// TIA Portal V18 export
DATA_BLOCK "HMI"   // DB1
{ S7_Optimized_Access := 'TRUE' }
VERSION : 0.1
// stored: AutoNumber true, DBAccessibleFromOPCUA true, IsOnlyStoredInLoadMemory false, IsRetainMemResEnabled false, IsWriteProtectedInAS false, MemoryReserve 100
   VAR
      "screen no to change" : Int;
      unit : Struct
         cm3 : Int;
         cm3_min : Int;
         ml : Int;
         ml_min : Int;
         "degree celsius" : Int;
         precentage : Int;
         seonds : Int;
         minutes : Int;
         hours : Int;
         bar : Int;
         mbar : Int;
         milliseconds : Int;
         RPM : Int;
         imp : Int;
         "cm3/r" : Int;
         set : Int;
         "real" : Int;
         "type" : Int;
         day : Int;
         "cm3/imp" : Int;
         "imp/rev" : Int;
         "m" : Int;
      END_STRUCT;
      "A" : Int;
      "B" : Int;
      "Screen no by function" : Int;
      "Current screen No" : Int;
      "Function ONS" : Struct
         "Dearing A" : Bool;
         "function deselected" : Bool;
         "Dearing B" : Bool;
         "Dearing A coil" : Bool;
         "dearing B Coil" : Bool;
         Flush : Bool;
         "pre run" : Bool;
         "Ratio Check" : Bool;
         "Shot metering Program" : Bool;
         "Continous metering prgram" : Bool;
         "metering program" : Bool;
         "recirculation A" : Bool;
         "recirculation B" : Bool;
         Recirculation : Bool;
         "pressure release A" : Bool;
         "pressure release B" : Bool;
         "Pressure release AB" : Bool;
         regeneration : Bool;
         "flush potlife" : Bool;
         "checkConditionA Coil" : Bool;
         "checkConditionB Coil" : Bool;
         checkConditionA : Bool;
         checkConditionB : Bool;
      END_STRUCT;
      "HMI User" : WString;
      AdminLogged : Bool;
      userlogged : Bool;
      "HMI user To hmi" : WString;
   END_VAR
   VAR RETAIN
      supplySelection : Int;
   END_VAR
BEGIN
END_DATA_BLOCK
